FUNCTION_BLOCK FloorIndicator (* Composite Function Block Type *)
  (* Standard: 61499-2 *)
  (* Version 0.0, 6/3/2016, Andrei, nxtControl GmbH, template *)
  PACKAGE Main;
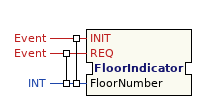
  EVENT_INPUT
    INIT WITH FloorNumber; (* Initialization Request *)
    REQ WITH FloorNumber; (* Normal Execution Request *)
  END_EVENT
  VAR_INPUT
    FloorNumber : INT; (* Input event qualifier *)
  END_VAR
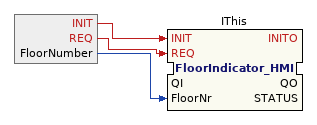
  FBS
    IThis : FloorIndicator_HMI;
  END_FBS
  EVENT_CONNECTIONS
    INIT TO IThis.INIT;
    REQ TO IThis.REQ;
  END_CONNECTIONS
  DATA_CONNECTIONS
    FloorNumber TO IThis.FloorNr;
  END_CONNECTIONS
END_FUNCTION_BLOCK
